{attribute 'qualified_only'}
VAR_GLOBAL
	// State cases
	caseInput : INT := 0;
	
	// Instruction string
	instructionString : STRING := 'Initializing lift';

	// General variables
	currentFloor : INT := 0;		// Holds the current floor
	targetFloor : INT := 0;			// The target floor
	liftMoving : BOOL := FALSE;		// Lift is moving
	liftDirection : BOOL := FALSE;	// Lift moving direction (1 is up, 0 is down)
	openDoor : BOOL := FALSE;		// True = open door, False = close door
	liftOperation : BOOL := FALSE;	// True = inside lift, False = outside lift
	
	 // Independent Door Task Control
    doorTask : BOOL := FALSE;         // Activate door task when lift reaches target floor
	
	// Buttons
	callLevel0 : BOOL := FALSE;		// Call base level
	callLevel1 : BOOL := FALSE;		// Call first level
	callLevel2 : BOOL := FALSE;		// Call second level
	setTargetLevel0 : BOOL := FALSE;
	setTargetLevel1 : BOOL := FALSE;
	setTargetLevel2 : BOOL := FALSE;

	// LEDs
	ledLevel0 : BOOL := FALSE;	// Set target floor to base floor
	ledLevel1 : BOOL := FALSE;	// Set target floor to first floor
	ledLevel2 : BOOL := FALSE;	// Set target floor to seocnd floor
	ledLiftMoving : BOOL := FALSE;
	ledDoorsOpen : BOOL := FALSE;
	
	// Time variables
	simulationTime : TON;			// Timer to simulate lift movement
	simulationPace : TIME := T#3S;	// Simulate lift movement (3 seconds)
    doorOpenPace : TIME := T#5S;      // Simulate door open duration (5 seconds)
END_VAR

(* stored: Version 1.1.0.1, ProductVersion 3.1.4024.12
   GVL GVL: Id {7b657eaf-3c50-4a66-b34e-94076662fc67} *)
